// TwinCAT 3 PLC project TCP_Client
// ProgramVersion: 3.1.4020.2
// libraries:
//   Tc2_Standard, * (Beckhoff Automation GmbH)
//   Tc2_System, * (Beckhoff Automation GmbH)
//   Tc2_TcpIp, * (Beckhoff Automation GmbH)
//   Tc3_Module, * (Beckhoff Automation GmbH)
// project tree:
//   DUTs/ E_State.TcDUT
//   / PlcTask.TcTTO
//   POUs/ FB_TcpClient.TcPOU, MAIN.TcPOU
// (motion and I/O tree: see PLC project tcp_server)
// real-time tasks:
//   TASK PlcTask: cycle T#10ms, priority 20, ADS port 350

CONFIGURATION TCP_Client
    RESOURCE PLC ON TwinCAT3
        TASK PlcTask(INTERVAL := T#10ms, PRIORITY := 20);
        PROGRAM MAIN WITH PlcTask : MAIN;
    END_RESOURCE
END_CONFIGURATION

// ---- DUTs/E_State.TcDUT
{attribute 'qualified_only'}
{attribute 'strict'}
TYPE E_State :
(
 	STATE_INIT,
	STATE_CONNECTING,
	STATE_RECEIVING_DATA,
	STATE_SENDING_DATA,
	STATE_PROCESSING_DATA
);
END_TYPE

// ---- POUs/MAIN.TcPOU
PROGRAM MAIN
VAR
	fbTcpClient		: FB_TcpClient;
	SrvNetId		: STRING := '';
	ServerAddress 	: STRING := '127.0.0.1';
	ServerPort 		: UDINT := 30000;
	
	sResponse		: STRING;
	sCommand		: STRING;
	bBusy			: BOOL;
	err				: BOOL;
	errid			: UDINT;
	
	bVar1			: BOOL;
	bVar2			: BOOL;
	test: STRING;
END_VAR

fbTcpClient(
	NetId:= SrvNetId, 
	ServerAdr:= ServerAddress, 
	ServerPort:= ServerPort, 
	sSend := sResponse,
	sReceive=> sCommand, 
	bBusy=> bBusy, 
	err=> err, 
	errid=> errid);
	
sResponse := sCommand;

IF sCommand = 'On1' THEN
	bVar1 := TRUE;
ELSIF sCommand = 'On2' THEN
	bVar2 := TRUE;
ELSE
	bVar1 := FALSE;
	bVar2 := FALSE;
END_IF

END_PROGRAM

// ---- POUs/FB_TcpClient.TcPOU
FUNCTION_BLOCK FB_TcpClient
VAR_INPUT
	NetId				: STRING; 	(* Server AmsNetId *)
	ServerAdr 			: STRING;	(* Server IP address *)
	ServerPort 			: UDINT;	(* Server port number *)
	sSend 				: STRING;	(* String to be sent *)
END_VAR
VAR_OUTPUT
	sReceive			: STRING;	(* String received *)
	bBusy				: BOOL;
	err					: BOOL;
	errid				: UDINT;
END_VAR
VAR
	fbSocketCloseAll	: FB_SocketCloseAll :=  ( sSrvNetID := '', tTimeout := DEFAULT_ADS_TIMEOUT );
	bCloseAll			: BOOL := TRUE;
		
	Timeout 			: TIME := T#10S;
	fbSocketConnect		: FB_SocketConnect;
	fbSocketReceive		: FB_SocketReceive;
	fbSocketAccept		: FB_SocketAccept;
	fbSocketSend 		: FB_SocketSend;
	hListen				: T_HSOCKET;
	hSocket				: T_HSOCKET;
    
	bConnAccepted		: BOOL;            	
	RxBuffer			: STRING;
	state				: E_State;
           	
	timer				: TON;
END_VAR

		
fbSocketConnect(
	sSrvNetId:= NetId, 
	sRemoteHost:= ServerAdr, 
	nRemotePort:= ServerPort, 
	bExecute:= , 
	tTimeout:= Timeout, 
	bBusy=> bBusy, 
	bError=> err, 
	nErrId=> errid,
	hSocket=> hSocket);
	
fbSocketSend(
		sSrvNetId:= NetId, 
		hSocket:= hSocket, 
		cbLen:= LEN(sSend), 
		pSrc:= ADR(sSend), 
		bExecute:= , 
		tTimeout:= Timeout, 
		bBusy=> bBusy, 
		bError=> err, 
		nErrId=> errid);

fbSocketReceive(
		sSrvNetId:= NetId, 
		hSocket:= hSocket, 
		cbLen:= SIZEOF(RxBuffer), 
		pDest:= ADR(RxBuffer), 
		bExecute:= , 
		tTimeout:= Timeout, 
		bBusy=> bBusy, 
		bError=> err, 
		nErrId=> errid, 
		nRecBytes=> );
		
CASE state OF
	E_State.STATE_INIT:
		//Open the port
		fbSocketConnect.bExecute := TRUE;
		state := E_State.STATE_CONNECTING;
		
		
	E_State.STATE_CONNECTING:
		fbSocketConnect.bExecute := FALSE;
		//Accept incoming connection every half a second
		IF NOT fbSocketConnect.bBusy AND NOT fbSocketConnect.bError THEN
			state := E_State.STATE_RECEIVING_DATA;
		END_IF
	
		
	E_State.STATE_RECEIVING_DATA:
		fbSocketReceive.bExecute := FALSE;
		
		IF NOT fbSocketReceive.bBusy AND NOT fbSocketReceive.bError THEN
			IF fbSocketReceive.nRecBytes = 0 THEN
				//if there's no data received, reset the fbSocketReceive
				fbSocketReceive.bExecute := TRUE;
			ELSE
				MEMSET(ADR(sReceive),0,SIZEOF(sReceive));
				MEMCPY(ADR(sReceive), fbSocketReceive.pDest, fbSocketReceive.nRecBytes);
				fbSocketSend.bExecute := TRUE;
				state := E_State.STATE_SENDING_DATA;
			END_IF
		END_IF
	
		
	E_State.STATE_SENDING_DATA:
		fbSocketSend.bExecute := FALSE;
		
		IF NOT fbSocketSend.bBusy AND NOT fbSocketSend.bError THEN 
				fbSocketReceive.bExecute := TRUE;
				state := E_State.STATE_RECEIVING_DATA;
		END_IF
END_CASE

END_FUNCTION_BLOCK
